METHOD M_InputMapping
VAR_INPUT
END_VAR
// TurnTable Axis sensor
arAxisCtrl_gb[AxisNo.TurnTable].SetupMode.bHomeSignal := NOT GVL_Input.uniDI.stDI.bTurnTable_Axis_HomeSensor;
// RoundBelt Axis sensor
arAxisCtrl_gb[AxisNo.RoundBelt].SetupMode.bHomeSignal := GVL_Input.uniDI.stDI.bRoundBelt_Axis_HomeSensor;
// Allocate Robot X Axis
arAxisCtrl_gb[AxisNo.Allocate_X].SetupMode.bPosLimitSignal:= NOT GVL_Input.uniDI.stDI.bAllocateRobot_Xaxis_PosLimit;
arAxisCtrl_gb[AxisNo.Allocate_X].SetupMode.bNegimitSignal:=  NOT GVL_Input.uniDI.stDI.bAllocateRobot_Xaxis_NegLimit;

//arAxisCtrl_gb[AxisNo.Allocate_Y].SetupMode.bHomeSignal:= ;
	//arAxisCtrl_gb[AxisNo.Allo cate_Y].SetupMode.bNegimitSignal:=;

arAxisCtrl_gb[AxisNo.OutRobot_X].SetupMode.bHomeSignal:= GVL_Input.uniDI.stDI.bOutRobot_Xaxis_HomeSensor;
arAxisCtrl_gb[AxisNo.OutRobot_X].SetupMode.bPosLimitSignal:=  NOT GVL_Input.uniDI.stDI.bOutRobot_Xaxis_PosLimit;
arAxisCtrl_gb[AxisNo.OutRobot_X].SetupMode.bNegimitSignal:=  NOT GVL_Input.uniDI.stDI.bOutRobot_Xaxis_NegLimit;

arAxisCtrl_gb[AxisNo.OutRobot_Y].SetupMode.bHomeSignal:= GVL_Input.uniDI.stDI.bOutRobot_Yaxis_HomeSensor;
arAxisCtrl_gb[AxisNo.OutRobot_Y].SetupMode.bPosLimitSignal:=  NOT GVL_Input.uniDI.stDI.bOutRobot_Yaxis_PosLimit;
arAxisCtrl_gb[AxisNo.OutRobot_Y].SetupMode.bNegimitSignal:=  NOT GVL_Input.uniDI.stDI.bOutRobot_Yaxis_NegLimit;

arAxisCtrl_gb[AxisNo.RackMotor].SetupMode.bNegimitSignal := NOT GVL_Input.uniDI.stDI.bStackPush_DCMotor_NegLimit;
arAxisCtrl_gb[AxisNo.RackMotor].SetupMode.bPosLimitSignal := not GVL_Input.uniDI.stDI.bStackPush_DCMotor_PosLimit;
END_METHOD

END_PROGRAM

// ---- Library/00_PackML/01_ObjectBase/FB_ModeBase_V1.TcPOU
(* the functionblock FB_ObjectBase_V1 is transmitted to every machineunit
*)
FUNCTION_BLOCK FB_ModeBase_V1 IMPLEMENTS ITF_UnitState
VAR_INPUT
    eModeCommand : DINT; //Mode from superior Unit
    eCommand     : E_PMLCommand := ePMLCommand_Abort; //Command for a new state from superior unit
	PackTag : Reference TO ST_PackMLv30;
END_VAR
VAR_OUTPUT
    eMode                  : DINT; //Actual mode of the Unit
    eState                 : E_PMLState (*:= ePMLState_Aborted*) ; //Actual state of the Unit
    bUndefinedDone         : BOOL; //When the SPS is started, the first state is Undefiend. bUndefined is TRUE, when the method Undefined has succesful finished
    bInvalidModeCommandOut : BOOL;
    bChangeIntoProduction  : BOOL;
END_VAR
VAR
    fbUnitModeManager : PML_UnitModeManager; //The PML_UnitModeManager manage the Modechanges
    fbStateMachine    : PML_StateMachine; //The PML_StateMachine mangae the Statechanges

    nStateModeChange : INT := 0; //Variable to handle the modechange
    nLastState       : E_PMLState; //Variable to store last state
END_VAR

CASE nStateModeChange OF
0:
	//Waiting for user request
	bChangeIntoProduction:= FALSE;
	IF  bButtonProductionReq AND (PackTag.Command.UnitMode = ePMLProtUnitMode_Production) AND (PackTag.Status.UnitModeCurrent = ePMLProtUnitMode_Invalid) THEN
			nStateModeChange	:= 1;
	ELSIF  PackTag.Command.UnitModeChangeRequest AND (PackTag.Command.UnitMode <> ePMLProtUnitMode_Production) THEN
			nStateModeChange	:= 1;
	ELSIF  bButtonProductionReq AND (PackTag.Command.UnitMode = ePMLProtUnitMode_Production) AND (PackTag.Status.UnitModeCurrent <> ePMLProtUnitMode_Production) THEN
			nStateModeChange	:= 3;
	END_IF
1:
	//Starting UnitModeManager 
	fbUnitModeManager.bExecute				:= TRUE;
	fbUnitModeManager.eModeCommand			:= eModeCommand;
	PackTag.Status.UnitModeChangeInProcess	:= TRUE;

	IF fbUnitModeManager.bDone THEN
		fbUnitModeManager.bExecute	:= FALSE;
		bInvalidModeCommandOut		:= FALSE;
		nStateModeChange			:= 0;
		bChangeIntoProduction		:= FALSE;
		
		PackTag.Status.UnitModeChangeInProcess	:= FALSE;
	ELSIF fbUnitModeManager.bError THEN
		bInvalidModeCommandOut		:= TRUE;
		fbUnitModeManager.bExecute	:= FALSE;
		
		nLastState					:= PackTag.Status.StateCurrent;
		nStateModeChange			:= 2;
		bChangeIntoProduction		:= FALSE;
		PackTag.Status.UnitModeChangeInProcess	:= FALSE;
	END_IF
2:
	//ErrorHanddling
	IF  PackTag.Command.UnitModeChangeRequest THEN
		nStateModeChange:=0;
		bInvalidModeCommandOut		:= FALSE;
	ELSIF nLastState<> PackTag.Status.StateCurrent THEN
		bInvalidModeCommandOut		:= FALSE;
	END_IF
	
3:
	//state to check, if command 'Porduction' is valid
	IF (PackTag.Status.StateCurrent = ePMLState_Aborted OR PackTag.Status.StateCurrent = ePMLState_Stopped OR PackTag.Status.StateCurrent = ePMLState_Idle) THEN
		bChangeIntoProduction		:= TRUE;
		IF stChangeIntoProduction.bYes OR stChangeIntoProduction.bYesReset THEN
			nStateModeChange			:= 1;		
		ELSIF stChangeIntoProduction.bNo THEN
			nStateModeChange			:= 0;
		END_IF
	ELSE
		nStateModeChange:= 2;
		bInvalidModeCommandOut		:= TRUE;
		nLastState					:= PackTag.Status.StateCurrent;
	END_IF
END_CASE


fbUnitModeManager(									
	eState			:= eState,
	eModeStatus		=> eMode,
	bDone			=> ,
	bError			=> ,
	nErrorId		=> );


IF fbUnitModeManager.eModeStatus <>  0 THEN
	//Calling the StateMachine, when there is a valid Mode
	fbStateMachine(
		eMode				:= eMode, 				
		eCommand			:= eCommand,			
		stSubUnitInfoRef	:= ,
		stOptions			:= , 
		eState				=> eState, 				
		bError				=> , 
		nErrorID			=> );
END_IF

//One of the methods is executing  by the actual state
CASE eState OF
	ePMLState_Undefined:
		M_Undefined();
	ePMLState_Clearing:
		M_Clearing();
	ePMLState_Stopped:
		M_Stopped();
	ePMLState_Starting:
		M_Starting();
	ePMLState_Idle:
		M_Idle();
	ePMLState_Suspended:
		M_Suspended();
	ePMLState_Execute:
		M_Execute();
	ePMLState_Stopping:
		M_Stopping();
	ePMLState_Aborting:
		M_Aborting();
	ePMLState_Aborted:
		M_Aborted();
	ePMLState_Holding:
		M_Holding();
	ePMLState_Held:
		M_Held();
	ePMLState_Unholding:
		M_Unholding();
	ePMLState_Suspending:
		M_Suspending();
	ePMLState_Unsuspending:
		M_Unsuspending();
	ePMLState_Resetting:
		M_Resetting();
	ePMLState_Completing:
		M_Completing();
	ePMLState_Complete:
		M_Complete();
END_CASE

{attribute 'object_name' := 'M_Aborted'}
METHOD M_Aborted
VAR_INPUT
END_VAR
M_StateComplete();
END_METHOD

{attribute 'object_name' := 'M_Aborting'}
METHOD M_Aborting
VAR_INPUT
END_VAR
M_StateComplete();
END_METHOD

{attribute 'object_name' := 'M_Clearing'}
METHOD M_Clearing
VAR_INPUT
END_VAR
M_StateComplete();
END_METHOD

{attribute 'object_name' := 'M_Complete'}
METHOD M_Complete
VAR_INPUT
END_VAR
M_StateComplete();
END_METHOD

{attribute 'object_name' := 'M_Completing'}
METHOD M_Completing
VAR_INPUT
END_VAR
M_StateComplete();
END_METHOD

{attribute 'object_name' := 'M_Execute'}
METHOD M_Execute
VAR_INPUT
END_VAR
M_StateComplete();
END_METHOD

{attribute 'object_name' := 'M_Held'}
METHOD M_Held
VAR_INPUT
END_VAR
M_StateComplete();
END_METHOD

{attribute 'object_name' := 'M_Holding'}
METHOD M_Holding
VAR_INPUT
END_VAR
M_StateComplete();
END_METHOD

{attribute 'object_name' := 'M_Idle'}
METHOD M_Idle
VAR_INPUT
END_VAR
M_StateComplete();
END_METHOD

{attribute 'object_name' := 'M_Resetting'}
METHOD M_Resetting
VAR_INPUT
END_VAR
M_StateComplete();
END_METHOD

{attribute 'object_name' := 'M_Starting'}
METHOD M_Starting
VAR_INPUT
END_VAR
M_StateComplete();
END_METHOD

{attribute 'object_name' := 'M_StateComplete'}
METHOD M_StateComplete
VAR_INPUT
END_VAR
//the actual state is completed
fbStateMachine.M_StateComplete();
END_METHOD

{attribute 'object_name' := 'M_Stopped'}
METHOD M_Stopped
VAR_INPUT
END_VAR
M_StateComplete();
END_METHOD

{attribute 'object_name' := 'M_Stopping'}
METHOD M_Stopping
VAR_INPUT
END_VAR
M_StateComplete();
END_METHOD

{attribute 'object_name' := 'M_Suspended'}
METHOD M_Suspended
VAR_INPUT
END_VAR
M_StateComplete();
END_METHOD

{attribute 'object_name' := 'M_Suspending'}
METHOD M_Suspending
VAR_INPUT
END_VAR
M_StateComplete();
END_METHOD

{attribute 'object_name' := 'M_Undefined'}
METHOD M_Undefined
VAR_INPUT
END_VAR
//bUndefinedDone := TRUE;
M_StateComplete();
END_METHOD

{attribute 'object_name' := 'M_Unholding'}
METHOD M_Unholding
VAR_INPUT
END_VAR
M_StateComplete();
END_METHOD

{attribute 'object_name' := 'M_Unsuspending'}
METHOD M_Unsuspending
VAR_INPUT
END_VAR
M_StateComplete();
END_METHOD

END_FUNCTION_BLOCK

// ---- Library/20_MachineUnits/21_StorageArea/Service/FB_LowerFeedInConveyor.TcPOU
FUNCTION_BLOCK FB_LowerFeedInConveyor EXTENDS FB_ActionBasic
VAR_INPUT
    xExecute    : BOOL;
    xAbort      : BOOL;
	xReset		: BOOL;
    Cylinder 	: REFERENCE TO UNI_CylinderList;
    TimeOut  	: LREAL := 30; // Unit : s
	Input		: ST_InputTable;
	OutPut		: ST_OutputTable;
	Motor		: REFERENCE TO UNI_MotorList;
END_VAR	
VAR_OUTPUT
    xAborted : BOOL;
    iErrorID : INT;
    ErrorMsg : T_MaxString;
END_VAR
VAR
    StateBehaviour   : CBML.ETrigATo;
    CurrentPosition : ST_PositionTable;
	uiCyclicStep    : UINT := 0;
	Reset_Rtrig 	:R_TRIG;
	
	TON_SensorDelay :TON;
	TON_ArrivedTimeOut :TON;
	TON_TimeOut :TON;
	fbExecuteEdgeDetect :FB_EdgeDetect;
END_VAR

THIS^.IBehaviourModel := StateBehaviour;
StateBehaviour(xExecute := xExecute,
              xAbort := xAbort OR fbExecuteEdgeDetect.xFallingEdge,
              udiTimeOut := LREAL_TO_UDINT( TimeOut*1000000),
              xDone => xDone,
              xBusy => xBusy,
              xError => xError,
              xAborted => xAborted);
//Error Mes
iErrorID := StateBehaviour._model.iErrorID;
ErrorMsg := M_GetErrorMsg(xErrorID := iErrorID);  

//Make sure that C# turns off execute to shut down the service
fbExecuteEdgeDetect(xInput :=xExecute);

//Reset 
Reset_Rtrig(CLK:= xReset);
IF Reset_Rtrig.Q THEN
	StateBehaviour.ResetModel(xCommit:=xReset);
END_IF

//Action
A00_BaseUnits();

ACTION A00_BaseUnits:
TON_SensorDelay(PT:= T#500MS);
TON_ArrivedTimeOut(PT:=T#30S);
TON_TimeOut(PT:=T#10S);
END_ACTION

METHOD CleanupAction
VAR_INPUT
    xAbortProposed : BOOL;
    iErrorIDProposed: INT;
END_VAR
VAR_OUTPUT
    xComplete : BOOL := TRUE;
    xAbort: BOOL := xAbortProposed;
 	iErrorID : INT := iErrorIDProposed;
END_VAR
END_METHOD

METHOD CyclicAction
VAR_INPUT
    itfTimingController : CBML.ITimingController;
END_VAR
VAR_OUTPUT
    xComplete : BOOL := TRUE;
    iErrorID : INT := 0;
END_VAR
xComplete :=FALSE;

CASE uiCyclicStep OF 
	
	100:	//檔盒上升， 呼叫輸送帶
		TON_TimeOut.IN:= TRUE;
		Cylinder.List.fbLowCV_Block2.M_Extend();
		IF Cylinder.List.fbLowCV_Block2.InFrontPosition THEN
			TON_TimeOut.IN:=FALSE;
			Motor.List.LowCV.M_MoveForward();
			uiCyclicStep:=150;
		END_IF
		IF TON_TimeOut.Q THEN 
			iErrorID :=10;
		END_IF
	150:	//check motor forward
		TON_TimeOut.IN :=TRUE;
		IF Motor.List.LowCV.InForWard THEN 
			TON_TimeOut.IN:=FALSE;
			uiCyclicStep:=200;
		END_IF
		IF TON_TimeOut.Q THEN
			iErrorID :=11;
		END_IF
	
	200:	//盒子到位, 延遲訊號,
		TON_ArrivedTimeOut.IN:= TRUE;
		TON_SensorDelay.IN := Input.bLowCV_Block2Detect_Sensor;
		IF TON_SensorDelay.Q THEN
			TON_SensorDelay.IN:=FALSE;
			TON_ArrivedTimeOut.IN:=FALSE;
			Cylinder.List.fbLowCV_Press4.M_Extend();
			uiCyclicStep:=300;
		END_IF
		IF TON_ArrivedTimeOut.Q THEN
			iErrorID :=9;
		END_IF
		
	300:	//檔盒下 等待第一盒到達最前sensor
		TON_TimeOut.IN:=TRUE;
		IF Cylinder.List.fbLowCV_Press4.InFrontPosition THEN
			Cylinder.List.fbLowCV_Block2.M_Retract();
		END_IF
		IF Cylinder.List.fbLowCV_Block2.InRearPosition THEN
			TON_TimeOut.IN:=FALSE;
			uiCyclicStep:=400;	
		END_IF
		IF TON_TimeOut.Q THEN
			iErrorID :=11;
		END_IF
		
	400:	//確認到最前sensor 
		TON_SensorDelay.IN:=Input.bLowCV_BoxArrived_Sensor;
		IF TON_SensorDelay.Q THEN
			TON_SensorDelay.IN:=FALSE;
			Cylinder.List.fbLowCV_Block2.M_Extend();
			uiCyclicStep:=500;
		END_IF
	
	500:	//釋放第二盒 
		IF 	Cylinder.List.fbLowCV_Block2.InFrontPosition THEN
			Cylinder.List.fbLowCV_Press4.M_Retract();
			uiCyclicStep:=600;
		END_IF
	600:	// 第二盒到檔盒位 第三盒壓盒檔上
		TON_SensorDelay.IN:= Input.bLowCV_Block2Detect_Sensor;
		IF TON_SensorDelay.Q THEN
			TON_SensorDelay.IN :=FALSE;
			Cylinder.List.fbLowCV_Press4.M_Extend();
			uiCyclicStep:= 700;
		END_IF
	
	700:	//釋放第二盒
		IF Cylinder.List.fbLowCV_Press4.InFrontPosition THEN
			Cylinder.List.fbLowCV_Block2.M_Retract();
			Cylinder.List.fbLowCV_Block1.M_Extend();
		END_IF
		IF Cylinder.List.fbLowCV_Block2.InRearPosition AND 
			Cylinder.List.fbLowCV_Block1.InFrontPosition THEN
			uiCyclicStep:= 800;
		END_IF
		
	800:	// 等待第二盒到夾盒位
		TON_SensorDelay.IN:=Input.bLowCV_Block1Detect_Sensor;
		IF TON_SensorDelay.Q THEN
			TON_SensorDelay.IN:=FALSE;
			Motor.List.LowCV.M_MotorStop();
			uiCyclicStep:=900;
		END_IF
	900:	//馬達停止 第一第二盒壓盒上
		IF Motor.List.LowCV.InStopped THEN
			Cylinder.List.fbLowCV_Press1.M_Extend();
			Cylinder.List.fbLowCV_Press2.M_Extend();
			Cylinder.List.fbLowCV_Block1.M_Retract();
			uiCyclicStep :=1000;
		END_IF
	1000:	//壓盒下
		IF Cylinder.List.fbLowCV_Press1.InFrontPosition AND 
			Cylinder.List.fbLowCV_Press2.InFrontPosition AND 
			Cylinder.List.fbLowCV_Block1.InRearPosition THEN
			Cylinder.List.fbLowCV_Press1.M_Retract();
			Cylinder.List.fbLowCV_Press2.M_Retract();
		END_IF
	1100:	//確認壓盒位置 回done
		IF Cylinder.List.fbLowCV_Press1.InRearPosition AND 
			Cylinder.List.fbLowCV_Press2.InRearPosition THEN 
			xComplete :=TRUE;
		END_IF
END_CASE
END_METHOD

METHOD ExitAction
VAR_INPUT
    xAfterCleanup : BOOL;
    xInCopyCode : BOOL;
END_VAR
TON_SensorDelay.IN:=FALSE;
END_METHOD

METHOD M_GetErrorMsg : T_MaxString
VAR_INPUT
	xErrorID: INT;
END_VAR

VAR
	
END_VAR
CASE xErrorID OF
	0:
		M_GetErrorMsg := 'No Error';
	1:
		M_GetErrorMsg := 'Action time out';
	2:
		M_GetErrorMsg := 'Position Data invalid';
	3:
		M_GetErrorMsg := 'LowCV_Block1 has Error in StartAction ';
	4:
		M_GetErrorMsg := 'LowCV_Block2 has Error in StartAction';
	5:
		M_GetErrorMsg := 'LowCV_Press1 has Error in StartAction';
	6:
		M_GetErrorMsg := 'LowCV_Press2 has Error in StartAction';
	7:
		M_GetErrorMsg := 'fbLowCV_Press3 has Error in StartAction';
	8:
		M_GetErrorMsg := 'fbLowCV_Press4 has Error in StartAction';
	9:
		M_GetErrorMsg := 'Box Arrived Time out not on LowCVBlock2' ;
	10:
		M_GetErrorMsg := 'Cylinder Error in CyclicAction';
	11:
		M_GetErrorMsg := 'Motor Error in CyclicAction';
									
		
		
		
		
END_CASE
END_METHOD

METHOD ResetAction
VAR_OUTPUT
    xComplete : BOOL := TRUE;
END_VAR
END_METHOD

METHOD StartAction
VAR_OUTPUT
    xComplete : BOOL := TRUE;
	iErrorID : INT := 0;
END_VAR
xComplete :=FALSE;

TON_SensorDelay.IN:=FALSE;

IF Cylinder.List.fbLowCV_Block1.xError THEN
	iErrorID := 3;
END_IF
IF Cylinder.List.fbLowCV_Block2.xError THEN
	iErrorID := 4;
END_IF
IF Cylinder.List.fbLowCV_Press1.xError THEN
	iErrorID := 5;
END_IF
IF Cylinder.List.fbLowCV_Press2.xError THEN
	iErrorID := 6;
END_IF
IF Cylinder.List.fbLowCV_Press3.xError THEN
	iErrorID := 7;
END_IF
IF Cylinder.List.fbLowCV_Press4.xError THEN
	iErrorID := 8;
END_IF

IF Cylinder.List.fbLowCV_Block1.InRearPosition AND
	Cylinder.List.fbLowCV_Block2.InRearPosition AND 
	Cylinder.List.fbLowCV_Press1.InRearPosition AND 
	Cylinder.List.fbLowCV_Press2.InRearPosition AND 
	Cylinder.List.fbLowCV_Press3.InRearPosition AND 
	Cylinder.List.fbLowCV_Press4.InRearPosition AND 
	Input.bLowCV_2ndBoxGap_Sensor THEN	//reverse logic sensor ,do make sure no box here 
	xComplete :=TRUE;
END_IF
END_METHOD

END_FUNCTION_BLOCK

// ---- Library/20_MachineUnits/22_AllocateArea/FB_AllocateAreaWithXPlanar.TcPOU
FUNCTION_BLOCK FB_AllocateAreaWithXPlanar EXTENDS FB_ModeBase_V1
VAR_INPUT
	
END_VAR
VAR_OUTPUT
END_VAR
VAR
	UnitInput :REFERENCE TO ST_AllocateInput;
	UnitOutput: REFERENCE TO ST_AllocateOutput;
END_VAR

{attribute 'object_name' := 'M_Aborted'}
METHOD M_Aborted 
VAR_INPUT
END_VAR
END_METHOD

{attribute 'object_name' := 'M_Aborting'}
METHOD M_Aborting
VAR_INPUT
END_VAR
END_METHOD

{attribute 'object_name' := 'M_Clearing'}
METHOD M_Clearing
VAR_INPUT
END_VAR
END_METHOD

{attribute 'object_name' := 'M_Complete'}
METHOD M_Complete
VAR_INPUT
END_VAR
END_METHOD

{attribute 'object_name' := 'M_Completing'}
METHOD M_Completing
VAR_INPUT
END_VAR
END_METHOD

{attribute 'object_name' := 'M_Execute'}
METHOD M_Execute
VAR_INPUT
END_VAR
M_StateComplete();
END_METHOD

{attribute 'object_name' := 'M_Held'}
METHOD M_Held
VAR_INPUT
END_VAR
END_METHOD

{attribute 'object_name' := 'M_Holding'}
METHOD M_Holding
VAR_INPUT
END_VAR
END_METHOD

{attribute 'object_name' := 'M_Idle'}
METHOD M_Idle
VAR_INPUT
END_VAR
END_METHOD

METHOD M_IOMapping
VAR_INPUT
END_VAR
//UnitInput := GVL_in
END_METHOD

{attribute 'object_name' := 'M_Resetting'}
METHOD M_Resetting
VAR_INPUT
END_VAR
END_METHOD

{attribute 'object_name' := 'M_Starting'}
METHOD M_Starting
VAR_INPUT
END_VAR
VAR
	uiStartingStep : DINT;
END_VAR
CASE eMode OF
    E_Mode.Auto:
        CASE uiStartingStep OF
            0: //
            1: //
            2: //
            3: //
            9900:
                M_StateComplete();
        END_CASE
END_CASE
END_METHOD

{attribute 'object_name' := 'M_Stopped'}
METHOD M_Stopped
VAR_INPUT
END_VAR
END_METHOD

{attribute 'object_name' := 'M_Stopping'}
METHOD M_Stopping
VAR_INPUT
END_VAR
END_METHOD

{attribute 'object_name' := 'M_Suspended'}
METHOD M_Suspended
VAR_INPUT
END_VAR
END_METHOD

{attribute 'object_name' := 'M_Suspending'}
METHOD M_Suspending
VAR_INPUT
END_VAR
END_METHOD

{attribute 'object_name' := 'M_Undefined'}
METHOD M_Undefined
VAR_INPUT
END_VAR
END_METHOD

{attribute 'object_name' := 'M_Unholding'}
METHOD M_Unholding
VAR_INPUT
END_VAR
END_METHOD

{attribute 'object_name' := 'M_Unsuspending'}
METHOD M_Unsuspending
VAR_INPUT
END_VAR
END_METHOD

END_FUNCTION_BLOCK

// ---- Library/99_Utilities/ErrorHandling/FB_ErrorHandler_OLD.TcPOU
{attribute 'reflection'}
FUNCTION_BLOCK PUBLIC FB_ErrorHandler_OLD IMPLEMENTS ITF_ErrorHandlerSubject
VAR_INPUT
END_VAR
VAR_OUTPUT
    astrActive : ARRAY [0..999] OF ST_Alarm_Tmax;	//State from all existing FB
	uiNumOfActError : UINT;	
	bErrorOccur 	:BOOL;
END_VAR
VAR
	
	//{attribute 'hide'}
	fbLocalSystemTime				: FB_LocalSystemTime := (bEnable := TRUE, dwCycle := 1);
    {attribute 'instance-path'} 
    {attribute 'noinit'}
    _strName: STRING(255); 					// Instance path of the FB for Diagnostic
			
	_stInfoState : ARRAY [1..GVL.MAX_Observer] OF ST_BehaviourInfo;	//State from all existing FB
	_stErrorState : ARRAY [1..GVL.MAX_Observer] OF BOOL;			//State from all existing FB
	_UniqueErrorCode : ARRAY [1..GVL.MAX_Observer] OF string;
	_uiNumberOfDevices : UINT;						//Number of Attached Devices
	uiHelp : INT; 									//Help Variable for Loop
	
	//Help Variables for Attaching and read Information from Devices
	aritfObserver : ARRAY [0..GVL.MAX_Observer]OF IBasicElement;
	uiLoop : UINT;
	uiErrorIndex : UINT;
    astrClear : ARRAY [0..999] OF ST_Alarm_Tmax;	//State from all existing FB
	_stErrorState_Clear : ARRAY [1..GVL.MAX_Observer] OF BOOL;			//State from all existing FB for clear	
	tonClearErrorDelay : TON;
	uiStep : UINT:=0;
	
END_VAR

_uiNumberOfDevices := 0;
fbLocalSystemTime();


tonClearErrorDelay(PT:=T#100MS);

CASE uiStep OF
	
0: //Init step
	tonClearErrorDelay.IN :=FALSE;
	bErrorOccur :=FALSE;
	uiStep :=100;
	
100: // Delay for a while
	tonClearErrorDelay.IN :=TRUE;
	IF tonClearErrorDelay.Q THEN
		uiStep := 300;
	END_IF
		
200: //Clear error
		astrActive := astrClear;
		_stErrorState :=_stErrorState_Clear;
		uiStep := 0;
300: //Working
FOR uiLoop := 0 TO GVL.MAX_Observer DO
    IF aritfObserver[uiLoop] <> 0 THEN

        _uiNumberOfDevices := _uiNumberOfDevices + 1;
        aritfObserver[uiLoop].GetModelState(
                xDone    => _stInfoState[uiLoop].xDone,
                xBusy    => _stInfoState[uiLoop].xBusy,
                xError   => _stInfoState[uiLoop].xError,
                xAborted => _stInfoState[uiLoop].xAborted,
                iErrorID => _stInfoState[uiLoop].iErrorID, 
				UniqueErrorCode =>_UniqueErrorCode[uiLoop]);

        _stInfoState[uiLoop].strName := aritfObserver[uiLoop].GetName();

        IF NOT _stErrorState[uiLoop] AND _stInfoState[uiLoop].xError THEN
            _stErrorState[uiLoop] := _stInfoState[uiLoop].xError;
			bErrorOccur :=TRUE;

            //Build Error String
            FOR uiHelp := 999 TO 0 BY -1 DO
                IF uiHelp > 0 THEN
                    // Sort the array down once, leaving the first row of the array empty.
                    astrActive[uiHelp] := astrActive[uiHelp - 1];
                ELSIF uiHelp = 0 THEN
                    astrActive[uiHelp].Message := CONCAT(
                            CONCAT(CONCAT('In FB ', _stInfoState[uiLoop].strName), ' the error is active : '),
                            FC_ErrorCode(_stInfoState[uiLoop].iErrorID));

                    astrActive[uiHelp].ID       := _stInfoState[uiLoop].iErrorID;
                    astrActive[uiHelp].Trigger  := _stInfoState[uiLoop].xError;
                    astrActive[uiHelp].DateTime := TIMESTRUCT_TO_PackMLTime(fbLocalSystemTime.systemTime);
					astrActive[uiHelp].UniqueErrorCode:=_UniqueErrorCode[uiLoop];
               		//astrActive[uiHelp].Value   :=	_UniqueErrorCode[uiLoop];
				 END_IF
            END_FOR
//        ELSIF _stErrorState[uiLoop] AND NOT _stInfoState[uiLoop].xError THEN
//            _stErrorState[uiLoop] := _stInfoState[uiLoop].xError;

//            //Build Error String
//            FOR uiHelp := 999 TO 0 BY -1 DO
//                IF uiHelp > 0 THEN
//                    astrActive[uiHelp] := astrActive[uiHelp - 1];
//                ELSIF uiHelp = 0 THEN
//                    astrActive[uiHelp].Message := CONCAT(
//                            CONCAT(CONCAT('In FB ', _stInfoState[uiLoop].strName), 'the following error is deactive:'),
//                            FC_ErrorCode(_stInfoState[uiLoop].iErrorID));
//                END_IF
//            END_FOR
        END_IF
		
	ELSE
	//	EXIT;	
    END_IF
END_FOR

END_CASE

METHOD AttachDevice 
(*Register a Device by the BehaiourModel Interface*)
VAR_INPUT
	(*Device which will be monitor from Error Handler*)
	IDevice	: IBasicElement;
END_VAR

VAR
	uiLoop: UINT;
END_VAR
FOR uiLoop := 1 TO GVL.MAX_Observer DO
	IF IDevice <> 0 AND THIS^.aritfObserver[uiLoop]= 0 THEN
		THIS^.aritfObserver[uiLoop] := IDevice;
		EXIT;
	END_IF
END_FOR
END_METHOD

METHOD ClearError
VAR_INPUT
END_VAR
astrActive := astrClear;
_stErrorState :=_stErrorState_Clear; // not necessary but keep it

uiStep := 200; // Go to clear error step
END_METHOD

METHOD DetachDevice 
(*Unregister a Device by the BehaiourModel Interface*)
VAR_INPUT
	(*Device which will be deleted from the monitor Error Handler list*)
	IDevice	: IBasicElement;
END_VAR

VAR
	uiLoop: UINT;
END_VAR
FOR uiLoop := 0 TO GVL.MAX_Observer DO
	IF IDevice <> 0 AND THIS^.aritfObserver[uiLoop]= IDevice THEN
		THIS^.aritfObserver[uiLoop] := 0;
		EXIT;
	END_IF
END_FOR
END_METHOD

END_FUNCTION_BLOCK

// ---- Library/99_Utilities/ErrorHandling/FB_ErrorHandler_abond.TcPOU
FUNCTION_BLOCK FB_ErrorHandler_abond EXTENDS FB_ActionBasic
VAR_INPUT
	xEnable : BOOL;
	stAdmin : REFERENCE TO ST_PMLa;
	AlarmList :REFERENCE TO ARRAY[0..999] OF ST_Alarm_Tmax;
END_VAR
VAR_OUTPUT
END_VAR
VAR
	StateBehavior : CBML.LConC;
	ErrorCount : DINT;
END_VAR

THIS^.IBehaviourModel := StateBehavior;
StateBehavior(xEnable:= xEnable, xBusy=> xBusy, xError=> xError);
//AlarmCtrl();
//IF btest THEN
//stAlarm.Trigger := TRUE;
//stAlarm.Message := 'test';
//AlarmCtrl.M_SetAlarm(stAdmin := GVL_Machine.PackTags[0].Admin, stAlarm := stAlarm);
//END_IF

METHOD CleanupAction
VAR_INPUT
    xAbortProposed : BOOL;
    iErrorIDProposed: INT;
END_VAR
VAR_OUTPUT
    xComplete : BOOL := TRUE;
    xAbort: BOOL := xAbortProposed;
 	iErrorID : INT := iErrorIDProposed;
END_VAR
END_METHOD

METHOD CyclicAction
VAR_INPUT
    itfTimingController : CBML.ITimingController;
END_VAR
VAR_OUTPUT
    xComplete : BOOL := TRUE;
    iErrorID : INT := 0;
END_VAR
VAR
	diCheckTriggerLoop : DINT;
	diCheckAlarmLoop : DINT;
	bHasSameID :BOOL;
END_VAR
VAR_INST
	diSearchID : DINT;
END_VAR
xComplete := FALSE;
bHasSameID := FALSE;
diSearchID := 0;
FOR diCheckTriggerLoop := 1 TO stAdmin.AlarmExtent DO
    IF stAdmin.Alarm[diCheckTriggerLoop].Trigger THEN
        FOR diCheckAlarmLoop := 0 TO 999 DO
            IF AlarmList[diCheckAlarmLoop].ID = stAdmin.Alarm[diCheckTriggerLoop].ID THEN
				diSearchID := diCheckTriggerLoop;
                bHasSameID := TRUE;
				EXIT;
            END_IF
        END_FOR
    END_IF

    IF NOT bHasSameID THEN
        ErrorCount := ErrorCount + 1;
        AlarmList[ErrorCount].ID := DINT_TO_UDINT(stAdmin.Alarm[diCheckTriggerLoop].ID);
        AlarmList[ErrorCount].Category := stAdmin.Alarm[diCheckTriggerLoop].Category;
        AlarmList[ErrorCount].Message := stAdmin.Alarm[diCheckTriggerLoop].Message;
        AlarmList[ErrorCount].Value := stAdmin.Alarm[diCheckTriggerLoop].Value;
        AlarmList[ErrorCount].Trigger := stAdmin.Alarm[diCheckTriggerLoop].Trigger;
    END_IF
END_FOR
END_METHOD

METHOD ExitAction
VAR_INPUT
    xAfterCleanup : BOOL;
    xInCopyCode : BOOL;
END_VAR
END_METHOD

METHOD ResetAction
VAR_OUTPUT
    xComplete : BOOL := TRUE;
END_VAR
END_METHOD

METHOD StartAction
VAR_OUTPUT
    xComplete : BOOL := TRUE;
	iErrorID : INT := 0;
END_VAR
END_METHOD

END_FUNCTION_BLOCK

// ---- Library/99_Utilities/ErrorHandling/FB_ErrorHandling.TcPOU
FUNCTION_BLOCK FB_ErrorHandling
VAR_INPUT
	xEnable : BOOL := TRUE;
	tInitBypassDelayTime : TIME;
END_VAR

VAR_OUTPUT
	xError		: BOOL; // Normal Error -> Go to Held
	//xFatalError : BOOL; // Fatal Error -> Go to Abort
	xWarning	: BOOL; // System have warning
	xSeverity : E_Severity;
END_VAR

VAR
	bFirstCycle			: BOOL := TRUE;
	bCoresysError		: BOOL; // At least one Coresys has an error 
	bXTSError			: BOOL; // At least one XTS has an error 
	dwXTSDiagNo			: DWORD; // XTS diag number
	strXTSDiagMessage : STRING(60); // XTS diag text
	uiXTSSeverity		: UINT; // XTS error severity
	bAppError			: BOOL; // User defined error
	bECatError			: BOOL; // EtherCAT module error
	dwAppDiagNo			: DWORD; // User diag number
	strAppDiagMessage : STRING(60); // User diag text
	uiAppErrSeverity	: UINT; // User error severity
	bSubsysError		: BOOL; // Subsys has an error
	// FB_AnyAborted_Rtrig : R_TRIG ;
	udiErrorCount					: UDINT;
	fbMachineCtrlInitDOne_Rtrig		: R_TRIG;
	fbMachineResetBtn_FTrig			: F_TRIG;
	bClearEthercatErr				: BOOL; // 臨時版本
	udiIndex						: UDINT;
	bAnySubAborted					: BOOL; // Currently, there is at least one Sub station in an aborted state.
	bST01_Alarm						: BOOL;
	bST03_Alarm						: BOOL;
	bST06_Alarm						: BOOL;
	bST10_Alarm						: BOOL;
	bST12_Alarm						: BOOL;
	bST14_Alarm						: BOOL;
	bST15_Alarm						: BOOL;
	bST17_Alarm						: BOOL;
	bST18_Alarm						: BOOL;
	bST20_Alarm						: BOOL;
	bST22_Alarm						: BOOL;
	bST23_Alarm						: BOOL;
	bST25_Alarm						: BOOL;
	bST27_Alarm						: BOOL;
	bST30_Alarm						: BOOL;
	bXTSShuttleError				: BOOL;
	bXTSModuleError					: BOOL;
	bXTSNcError						: BOOL;
	bResetRetry						: BOOL;
	TON_ResetRetry					: TON;
	FB_CoresysErrorHandler			: FB_CoresysErrorHandler;
	TON_ClearDelayCheck				: TON;
	bSubsysWarning					: BOOL;
	Ton_InitBypassDelay				: TON;
	FB_EtherCATErrorHandler			: FB_EtherCATErrorHandler;
	arrUnitsWarningHandler			: ARRAY[1..cudiXTS_MaxIndex]OF FB_AppWarningHandler;
	I_UnitsWarningHandler			: ARRAY[1..cudiXTS_MaxIndex]OF ITF_SubUnitWarning;
	TON_KeepMDSError 				: TON;
	TON_CheckMDSNoError				: TON;
	bCheckMDSError					: BOOL;
	TOF_KeepMDSError_Delay			: TOF;

END_VAR

Ton_InitBypassDelay(PT:= T#5S);
IF NOT xEnable THEN
	RETURN;
ELSIF ( bFirstCycle = TRUE ) THEN
	Ton_InitBypassDelay.IN := TRUE;
	M_OneTimeInit();
	RETURN;
END_IF


//TON_ClearDelayCheck(IN := bClearbyPassDelay, PT := T#800MS);

//IF TON_ClearDelayCheck.Q THEN
//	bClearbyPassDelay := FALSE;
//END_IF

//IF bReset_gb THEN
//	THIS^.M_Reset();
//END_IF
//IF   NOT FB_Safety.bSafetyOK AND_THEN M_FindMDSError() THEN
//	bKeepMDSError := TRUE;
//END_IF
//TON_KeepMDSError(IN := bKeepMDSError,PT := T#3S);
//bCheckMDSError := FALSE;
//FOR udiIndex := 1 TO UDINT_TO_UINT(udiMax_MachineAlarm_Index) DO
//	IF PackTags.Machine.Admin.Alarm[udiIndex].ID = DINT#990281 THEN
//		bCheckMDSError := TRUE;
//	END_IF
//END_FOR
//TON_CheckMDSNoError(IN := (NOT FB_MDS.bMoverIdDetectionError) AND (NOT FB_MDS.bError) AND (NOT bCheckMDSError), PT := T#1S  );
//TOF_KeepMDSError_Delay(IN:= TON_CheckMDSNoError.Q ,PT:=T#2S);

//IF  TOF_KeepMDSError_Delay.Q THEN
//	bKeepMDSError := false;
//END_IF
// Alarm Histroy Upload
M_UploadData();
//------------------------------------------------------------------------------------------------------
//------------------------------------- Scan errors  ---------------------------------------------------  
//------------------------------------------------------------------------------------------------------
M_ScanError();

M_ErrorAction(xSeverity=> xSeverity);

ACTION EtherCAT_Diag:
fbMachineCtrlInitDOne_Rtrig(CLK := bMachineCtrlInitDOne);
fbMachineResetBtn_FTrig(CLK := bReset_gb);

IF fbMachineCtrlInitDOne_Rtrig.Q OR fbMachineResetBtn_FTrig.Q THEN
	FOR udiIndex := 1 TO TO_UDINT(udiECatMasterNum) DO
		// Check mapping status
		IF (F_GetMappingStatus(p := ADR(arruiFrm0WcStateMapping[udiIndex]), n := SIZEOF(arruiFrm0WcStateMapping[udiIndex]))
			= EPlcMappingStatus.MS_Mapped)
			OR (
			F_GetMappingStatus(p := ADR(arruiFrm0WcStateMapping[udiIndex]), n := SIZEOF(arruiFrm0WcStateMapping[udiIndex]))
			= EPlcMappingStatus.MS_Partial)
			THEN
			arrfbEtherCatDiagnostics[udiIndex].bEnable := TRUE;
		END_IF
	END_FOR
END_IF

// 臨時版本
IF bClearEthercatErr THEN
	FOR udiIndex := 1 TO TO_UDINT(udiECatMasterNum) DO
		// Check mapping status
		IF (F_GetMappingStatus(p := ADR(arruiFrm0WcStateMapping[udiIndex]), n := SIZEOF(arruiFrm0WcStateMapping[udiIndex]))
			= EPlcMappingStatus.MS_Mapped)
			OR (
			F_GetMappingStatus(p := ADR(arruiFrm0WcStateMapping[udiIndex]), n := SIZEOF(arruiFrm0WcStateMapping[udiIndex]))
			= EPlcMappingStatus.MS_Partial)
			THEN
			arrfbEtherCatDiagnostics[udiIndex].bEnable := FALSE;
		END_IF
	END_FOR

	bClearEthercatErr := FALSE;
END_IF

// FB_EtherCatDiagnostics
FOR udiIndex := 1 TO TO_UDINT(udiECatMasterNum) DO
	// Check mapping status
	IF (F_GetMappingStatus(p := ADR(arruiFrm0WcStateMapping[udiIndex]), n := SIZEOF(arruiFrm0WcStateMapping[udiIndex]))
		= EPlcMappingStatus.MS_Mapped)
		OR (F_GetMappingStatus(p := ADR(arruiFrm0WcStateMapping[udiIndex]), n := SIZEOF(arruiFrm0WcStateMapping[udiIndex]))
		= EPlcMappingStatus.MS_Partial)
		THEN
		arrfbEtherCatDiagnostics[udiIndex](uiFrm0WcStateMapping := arruiFrm0WcStateMapping[udiIndex],
											uiFrm1WcStateMapping := arruiFrm1WcStateMapping[udiIndex],
											uiFrm2WcStateMapping := arruiFrm2WcStateMapping[udiIndex],
											uiFrm3WcStateMapping := arruiFrm3WcStateMapping[udiIndex],
											wDeviceIDMapping := arrwDeviceIDMapping[udiIndex],
											bEnable :=,
											pstDiagnosticResult := ADR(arrstDiagnosticResult[udiIndex]),
											pstFuncBlocksErr := ADR(arrstFuncBlocksErr[udiIndex]),
											bBusy =>,
											bActive =>,
											bError =>);
	END_IF
END_FOR
END_ACTION

METHOD FB_exit : BOOL
VAR_INPUT
	bInCopyCode : BOOL; // if TRUE, the exit method is called for exiting an instance that is copied afterwards (online change).
END_VAR
// 避免再切config時出現動態記憶體異常
fbAlarmTrigList.releaseQueue();
fbAlarmResetList.releaseQueue();
END_METHOD

METHOD GetAbort : BOOL
VAR_INPUT
END_VAR
VAR
	// Subsys Station number
	udiSubIndex : UDINT;
END_VAR
VAR_OUTPUT
	xErrorID : UDINT;
	//	ErrorMsg: STRING(255);
END_VAR
GetAbort := FALSE;

FOR udiSubIndex := 1 TO cudiXTS_MaxIndex DO
	IF (PackTags.arrSubSys_Station^[udiSubIndex].Status.StateCurrent = ePMLState_Aborted)
		AND (stSysParameters_Current.arIndexProductionValid[udiSubIndex] = E_ProductionValid.Valid)
		THEN
		xErrorID := 1100 + udiSubIndex;
		//FB_AppErrorHandler.M_SetAlarm(xUnitName := FB_AppErrorHandler.GetName(), xErrorID := xErrorID);
		GetAbort := TRUE;
		RETURN;

	END_IF
END_FOR

IF (PackTags.XTS.Status.StateCurrent = ePMLState_Aborted) THEN
	xErrorID := 1100;
	//FB_AppErrorHandler.M_SetAlarm(xUnitName := FB_AppErrorHandler.GetName(), xErrorID := xErrorID);
	GetAbort := TRUE;
END_IF
END_METHOD

METHOD GetHeld : BOOL
VAR_INPUT
END_VAR
VAR
	// Subsys Station number
	udiSubIndex : UDINT;
END_VAR
GetHeld := FALSE;

FOR udiSubIndex := 1 TO cudiXTS_MaxIndex DO
	IF (PackTags.arrSubSys_Station^[udiSubIndex].Status.StateCurrent = ePMLState_Held) THEN
		GetHeld := TRUE;
	END_IF
END_FOR

IF (PackTags.XTS.Status.StateCurrent = ePMLState_Held) THEN
	GetHeld := TRUE;
END_IF
END_METHOD

METHOD M_CoresysErrorHandle
VAR_INPUT
END_VAR
VAR
	udiLoop : UDINT;
	xarObserver		: ARRAY[1..MAX_Observer] OF ST_Alarm;
END_VAR
VAR_INST
	xErrorFound : BOOL;
END_VAR
VAR_OUTPUT
	xError : BOOL;
END_VAR
//IF bMachineCtrlInitDOne THEN
	FB_CoresysErrorHandler(xError=>xError);
//END_IF
END_METHOD

METHOD M_ErrorAction
VAR_INPUT
END_VAR

VAR
	udiLoop: UDINT;
END_VAR
VAR_INST
	bSafetyDoorOpened : BOOL;
END_VAR
VAR_OUTPUT
	xSeverity : E_Severity;
END_VAR
//xSeverity := 0;
//FOR udiLoop := 1 TO udiMax_MachineAlarm_Index DO
//	IF PackTags.Machine.Admin.Alarm[udiLoop].Value > xSeverity THEN
//		xSeverity := PackTags.Machine.Admin.Alarm[udiLoop].Value;
//	END_IF
//END_FOR
//bSafetyDoorOpened := FALSE;
//FOR udiLoop := 1 TO cgudiNumOfSafetyDoor DO
//	IF arrSafetyDoorStatus[udiLoop].bButton THEN
//		bSafetyDoorOpened := TRUE;
//		EXIT;
//	END_IF
//END_FOR
//IF ( xSeverity = E_Severity.Level7 ) THEN
//	IF xError
//		AND NOT ((PackTags.Machine.Status.StateCurrent=ePMLState_Aborted) 
//		OR (PackTags.Machine.Status.StateCurrent=ePMLState_Aborting) 
//		OR (PackTags.Machine.Status.StateCurrent = ePMLState_Clearing))
//	THEN
//		PackTags.Machine.Command.CntrlCmd := ePMLCommand_Abort;
//		PackTags.Machine.Command.CmdChangeRequest := TRUE;
//	END_IF
//ELSIF xSeverity = E_Severity.Level6 THEN
//	IF xError THEN
//		IF (PackTags.Machine.Status.StateCurrent= ePMLState_Execute AND NOT ((PackTags.Machine.Status.UnitModeCurrent = E_MachineMode.Manual) AND bSafetyDoorOpened) )
//			OR  (PackTags.Machine.Status.StateCurrent= ePMLState_Suspended)
//			OR  (PackTags.Machine.Status.StateCurrent= ePMLState_Unsuspending)
//			OR  (PackTags.Machine.Status.StateCurrent= ePMLState_Suspending)
//			OR  (PackTags.Machine.Status.StateCurrent= ePMLState_Held)
//			OR  (PackTags.Machine.Status.StateCurrent= ePMLState_Unholding)
//			OR  (PackTags.Machine.Status.StateCurrent= ePMLState_Holding) 
//		THEN
//		PackTags.Machine.Command.CntrlCmd := ePMLCommand_Hold;
//		PackTags.Machine.Command.CmdChangeRequest := TRUE;
//		ELSIF (PackTags.Machine.Status.UnitModeCurrent = E_MachineMode.Manual) AND bSafetyDoorOpened
//				AND NOT FB_MDS.bAllShuttlesNotMoving
////				AND NOT (PackTags.XTS.Status.StateCurrent = ePMLState_Aborted)
////				AND NOT (PackTags.XTS.Status.StateCurrent = ePMLState_Aborting)
////				AND NOT (PackTags.XTS.Status.StateCurrent = ePMLState_Clearing)
//		THEN
//		PackTags.XTS.Command.CntrlCmd := ePMLCommand_Abort;
//		PackTags.XTS.Command.CmdChangeRequest := TRUE;
//		END_IF
//	END_IF
//ELSIF xSeverity = E_Severity.Level5 THEN
//	IF xError THEN
//		IF (PackTags.Machine.Status.StateCurrent= ePMLState_Execute)
//			AND (PackTags.Machine.Status.UnitModeCurrent = E_MachineMode.Initialization)
//		THEN
//		PackTags.Machine.Command.CntrlCmd := ePMLCommand_Stop;
//		PackTags.Machine.Command.CmdChangeRequest := TRUE;
//		END_IF
//	END_IF
//END_IF
END_METHOD

METHOD M_EtherCATErrorHandler
VAR_INPUT
END_VAR
VAR_OUTPUT
	xError:BOOL;
END_VAR
//THIS^.xError := FALSE;
FOR udiIndex := 1 TO udiECatMasterNum DO
	arFB_ECatDiag[udiIndex](udiEcDeviceIndex:=udiIndex,xError=>);
	IF arFB_ECatDiag[udiIndex].xError THEN
		xError :=TRUE;
	END_IF
END_FOR
END_METHOD

METHOD M_FindMDSError : BOOL
VAR_INPUT
END_VAR
VAR
	udiAlarmIndex : UDINT;
END_VAR
FOR udiAlarmIndex := 1 TO udiMax_MachineAlarm_Index DO
	IF PackTags.Machine.Admin.Alarm[udiAlarmIndex].ID = DINT#990281 THEN
		M_FindMDSError := TRUE;
	END_IF
END_FOR
END_METHOD

METHOD M_OneTimeInit
VAR_INPUT
END_VAR

IF Ton_InitBypassDelay.Q THEN
	bFirstCycle := FALSE;
	Ton_InitBypassDelay.IN := FALSE;
END_IF
END_METHOD

METHOD M_Reset
VAR_INPUT
END_VAR
//// Clear Safety error.
//IF FB_Safety.stSafetyMapping.stSafetyProject.stGroupInput.bInRun
//	AND NOT bEStopActived_gb THEN
//	FB_Safety.reset();
//END_IF

//// XTS motion calculation
//IF fbXTSCalc.bError THEN
//	fbXTSCalc.M_Reset();
//END_IF


//IF FB_XTS.FB_InitializationMode.xError THEN
//	FB_XTS.FB_InitializationMode.M_ClearStatus();
//END_IF

//IF fbShuttlesConsvNGMon.bError THEN
//	fbShuttlesConsvNGMon.M_Reset();
//END_IF



//IF FB_CoreSys_gb.FB_Machine_ProductionMode.xError THEN
//	FB_CoreSys_gb.FB_Machine_ProductionMode.M_ClearError();
//END_IF


//IF FB_CoreSys_gb.FB_Machine_InitializationMode.xError THEN
//	FB_CoreSys_gb.FB_Machine_InitializationMode.M_ClearError();
//END_IF


//IF FB_LubricationCamPnp.Error THEN
//	FB_LubricationCamPnp.Reset();
//END_IF

//IF FB_LubricationXTS.Error THEN
//	FB_LubricationXTS.Reset();
//END_IF
	

//IF FB_HealthBit_HMI.bError THEN
//	FB_HealthBit_HMI.M_Reset();
//END_IF

//IF FB_IPCShutDown.bError THEN
//	FB_IPCShutDown.M_Reset();
//END_IF 		

//IF FB_IPCPowerFailureHandler.bError THEN
//	FB_IPCPowerFailureHandler.M_Reset();
//END_IF

//IF FB_Reset_Rtrig.Q AND FB_DataRecovery.bError THEN
//	FB_DataRecovery.M_Reset();
//END_IF 

//IF FB_Reset_Rtrig.Q AND fbTerminateBatch.bError THEN
//	fbTerminateBatch.M_Reset();
//END_IF

//IF bECatError THEN
//	bECatError := FALSE;
//END_IF
END_METHOD

METHOD M_ScanError
VAR_INPUT
END_VAR

VAR
	udiLoop : UDINT;
END_VAR
VAR_INST
	bECatError_Mem : BOOL;
END_VAR
// Ethercat Diag
EtherCAT_Diag();
//FB_EtherCATErrorHandler(xError=>bECatError);
M_EtherCATErrorHandler(xError =>bECatError_Mem);
IF  bECatError_Mem THEN
	bECatError := TRUE;
END_IF
// XTS error combinations.
M_XTSErrorHandle();

// Coresys error combinations.
M_CoresysErrorHandle(xError=> bAppError);
bCoresysError := bXTSError OR bAppError OR bECatError;

// Subsys error combinations

M_SubsysErrorHandle(xError => bSubsysError);
//M_SubsysWarrningHandle(xWarning => bSubsysWarning);
M_SubsysWarningHandler();
//------------------------------------------------------------------------------------------------------
//------------------------------ Calculate global error flag  ------------------------------------------  
//------------------------------------------------------------------------------------------------------
xError := bCoresysError OR bSubsysError;
xWarning := bSubsysWarning;
END_METHOD

METHOD M_SubsysErrorHandle
VAR_INPUT
END_VAR
VAR
	udiLoop : UDINT;
END_VAR
VAR_OUTPUT
	xError : BOOL;
END_VAR
IF bMachineCtrlInitDOne THEN
	FOR udiLoop := 1 TO cudiXTS_MaxIndex DO
		IF arAlarmHandleValid[udiLoop] = E_AlarmHandleValid.Valid THEN
			arFB_SubsysErrorScan[udiLoop](xSubPMLa := PackTags.arrSubSys_Station^[udiLoop].Admin,
										xUnitName := CONCAT('ST', UDINT_TO_STRING(udiLoop)),
										xUnitID := UDINT_TO_DINT(udiLoop));
		END_IF
	END_FOR
END_IF

bST01_Alarm := (arFB_SubsysErrorScan[1].uiCurrentAlarmsCount > 0);
bST03_Alarm := (arFB_SubsysErrorScan[3].uiCurrentAlarmsCount > 0);
bST06_Alarm := (arFB_SubsysErrorScan[6].uiCurrentAlarmsCount > 0);
bST10_Alarm := (arFB_SubsysErrorScan[10].uiCurrentAlarmsCount > 0);
bST12_Alarm := (arFB_SubsysErrorScan[12].uiCurrentAlarmsCount > 0);
bST14_Alarm := (arFB_SubsysErrorScan[14].uiCurrentAlarmsCount > 0);
bST15_Alarm := (arFB_SubsysErrorScan[15].uiCurrentAlarmsCount > 0);
bST17_Alarm := (arFB_SubsysErrorScan[17].uiCurrentAlarmsCount > 0);
bST18_Alarm := (arFB_SubsysErrorScan[18].uiCurrentAlarmsCount > 0);
bST20_Alarm := (arFB_SubsysErrorScan[20].uiCurrentAlarmsCount > 0);
bST22_Alarm := (arFB_SubsysErrorScan[22].uiCurrentAlarmsCount > 0);
bST23_Alarm := (arFB_SubsysErrorScan[23].uiCurrentAlarmsCount > 0);
bST25_Alarm := (arFB_SubsysErrorScan[25].uiCurrentAlarmsCount > 0);
bST27_Alarm := (arFB_SubsysErrorScan[27].uiCurrentAlarmsCount > 0);
bST30_Alarm := (arFB_SubsysErrorScan[30].uiCurrentAlarmsCount > 0);

xError := bST01_Alarm
	OR bST03_Alarm
	OR bST06_Alarm
	OR bST10_Alarm
	OR bST12_Alarm
	OR bST14_Alarm
	OR bST15_Alarm
	OR bST17_Alarm
	OR bST18_Alarm
	OR bST20_Alarm
	OR bST22_Alarm
	OR bST23_Alarm
	OR bST25_Alarm
	OR bST27_Alarm
	OR bST30_Alarm;
END_METHOD

METHOD M_SubsysWarningHandler
VAR_INPUT
END_VAR

VAR
	udiLoop: UDINT;
END_VAR
IF bMachineCtrlInitDOne THEN
	FOR udiLoop := 1 TO cudiXTS_MaxIndex DO
		arrUnitsWarningHandler[udiLoop]();
		IF arAlarmHandleValid[udiLoop] = E_AlarmHandleValid.Valid THEN
			I_UnitsWarningHandler[udiLoop] := arrUnitsWarningHandler[udiLoop];
			I_UnitsWarningHandler[udiLoop].SetUnitWarningList := (PackTags.arrSubSys_Station^[udiLoop].Admin.Warning );
			I_UnitsWarningHandler[udiLoop].SetUnitID := UDINT_TO_DINT(udiLoop);
			I_UnitsWarningHandler[udiLoop].SetUnitName := CONCAT('ST', UDINT_TO_STRING(udiLoop));
		END_IF
	END_FOR
	bSubsysWarning := FALSE;
	FOR udiLoop := 1 TO cudiXTS_MaxIndex DO
		IF arAlarmHandleValid[udiLoop] = E_AlarmHandleValid.Valid THEN
			IF  I_UnitsWarningHandler[udiLoop].GetWarningStatus THEN
				bSubsysWarning := TRUE;
			END_IF
		END_IF
	END_FOR
END_IF
END_METHOD

METHOD M_SubsysWarrningHandle
VAR_INPUT
END_VAR

VAR
	udiLoop : UDINT;
END_VAR
VAR_INST
	bST30_EmphtyCheck_NG1 : BOOL;
	bST30_EmphtyCheck_NG2 : BOOL;
	bST30_EmphtyCheck_NG3 : BOOL;
	bST30_EmphtyCheck_NG4 : BOOL;
END_VAR
VAR_OUTPUT
	xWarning : BOOL;
END_VAR
IF bMachineCtrlInitDOne THEN
//	FOR udiLoop := 1 TO cudiXTS_MaxIndex DO
//		IF arAlarmHandleValid[udiLoop] = E_AlarmHandleValid.Valid THEN
//			arFB_WarrningHandler[udiLoop](xSubPMLa := PackTags.arrSubSys_Station^[udiLoop].Admin,
//											xUnitName := CONCAT('ST', UDINT_TO_STRING(udiLoop)),
//											xUnitID := UDINT_TO_DINT(udiLoop));
//		END_IF
//	END_FOR
END_IF

bST30_EmphtyCheck_NG1 := FUN_ObserverWarning(xErrorID := 200, xUnitID := 30);
bST30_EmphtyCheck_NG2 := FUN_ObserverWarning(xErrorID := 201, xUnitID := 30);
bST30_EmphtyCheck_NG3 := FUN_ObserverWarning(xErrorID := 202, xUnitID := 30);
bST30_EmphtyCheck_NG4 := FUN_ObserverWarning(xErrorID := 203, xUnitID := 30);
END_METHOD

METHOD M_UploadData
VAR_INPUT
END_VAR
M_UploadTriggerData();
M_UploadResetData();
END_METHOD

METHOD PRIVATE M_UploadResetData : BOOL
VAR_INPUT
END_VAR
VAR_INST
	iStep : INT;
	stAlarm	: ST_Alarm_WString;
	stAlarmInf_DB: ST_AlarmInfo_DB;
END_VAR
CASE iStep OF
	0:
		IF 			fbAlarmResetList.udiGetQueuedAmount <> 0 // Queue裡面有資料
		AND_THEN 	fbAlarmResetList.readElementbyIndex(udiIndex := 1,	pbtReadElement := ADR(stAlarm),	udiReadSize := SIZEOF(stAlarm),	uiErrorID =>) THEN
			
			iStep := iStep + 100;
		END_IF
	
	100:
		stAlarmInf_DB.diMsgNumber := stAlarm.ID;
		stAlarmInf_DB.iMsgClass := stAlarm.eMsgClass;
		stAlarmInf_DB.iMsgProc := 1;
		stAlarmInf_DB.iStateAfter := 0;
		stAlarmInf_DB.sPLC := 'CoreSystem';
		stAlarmInf_DB.sTimeString := FUN_DateTime_To_TMaxString(DateTime := stAlarm.ackDateTime);
		stAlarmInf_DB.wsMsgText := stAlarm.Message;
		
		IF NOT Global_DataFlow.bDataFlowTestByLeo THEN
			IF FB_DataUpload.M_AddAlarmHistory(stAlarmInfo := stAlarmInf_DB) THEN
				iStep := iStep + 100;
			END_IF
		ELSE
			(* Add alarm history to database *)
//			IF Global_DataFlow.fbDataBaseManagement.M_Add_AlarmHistory(addData := stAlarmInf_DB) THEN
//				iStep := iStep + 100;
//			END_IF
		END_IF
	
	200:
		IF fbAlarmResetList.dequeueElement(pbtDequeueElement := ADR(stAlarm),
														udiDequeueSize := SIZEOF(stAlarm),
														uiErrorID =>)
			THEN // 清除已經上傳的資料
			iStep := 0;
		END_IF
		
END_CASE
END_METHOD

METHOD PRIVATE M_UploadTriggerData : BOOL
VAR_INPUT
END_VAR
VAR_INST
	iStep : INT;
	stAlarm	: ST_Alarm_WString;
	stAlarmInf_DB: ST_AlarmInfo_DB;
END_VAR
CASE iStep OF
	0:
		IF 			fbAlarmTrigList.udiGetQueuedAmount <> 0 // Queue裡面有資料
		AND_THEN 	fbAlarmTrigList.readElementbyIndex(udiIndex := 1,	pbtReadElement := ADR(stAlarm),	udiReadSize := SIZEOF(stAlarm),	uiErrorID =>) THEN
			
			iStep := iStep + 100;
		END_IF
	
	100:
		stAlarmInf_DB.diMsgNumber := stAlarm.ID;
		stAlarmInf_DB.iMsgClass := stAlarm.eMsgClass;
		stAlarmInf_DB.iMsgProc := 1;
		stAlarmInf_DB.iStateAfter := 1;
		stAlarmInf_DB.sPLC := 'CoreSystem';
		stAlarmInf_DB.sTimeString := FUN_DateTime_To_TMaxString(DateTime := stAlarm.DateTime);
		stAlarmInf_DB.wsMsgText := stAlarm.Message;
		
		IF NOT Global_DataFlow.bDataFlowTestByLeo THEN
			IF FB_DataUpload.M_AddAlarmHistory(stAlarmInfo := stAlarmInf_DB) THEN
				iStep := iStep + 100;
			END_IF
		ELSE
			IF Global_DataFlow.fbDataBaseManagement.M_Add_AlarmHistory(addData := stAlarmInf_DB) THEN
				iStep := iStep + 100;
			END_IF
		END_IF
		
	200:
		IF fbAlarmTrigList.dequeueElement(pbtDequeueElement := ADR(stAlarm),
														udiDequeueSize := SIZEOF(stAlarm),
														uiErrorID =>)
			THEN // 清除已經上傳的資料
			iStep := 0;
		END_IF
		
END_CASE
END_METHOD

METHOD M_XTSErrorHandle
VAR_INPUT
END_VAR
FB_XTSErrorHandler(xSubPMLa := PackTags.XTS.Admin, xUnitName := 'XTS', xUnitID := 99,xError=>bXTSError);
END_METHOD

END_FUNCTION_BLOCK

// ---- Library/99_Utilities/FB_XY_Move.TcPOU
(* This FB is use to controll two axis to gear in move at the same time 
*)
FUNCTION_BLOCK FB_XY_Move EXTENDS FB_ActionBasic
VAR_INPUT
	xExecute : BOOL;
	xAbort : BOOL;
	xReset :BOOL;
	AxisX_No : AxisNo;
	AxisY_No : AxisNo;
	
    TimeOut     : LREAL := 30; // Unit : s
END_VAR
VAR_OUTPUT
	xAborted : BOOL;
END_VAR
VAR
	StateBehavior : CBML.ETrigATo;
	CurrentPosData :ST_PositionTable;
	uiCyclicStep :UINT;
END_VAR

THIS^.IBehaviourModel := StateBehavior;
StateBehavior(xExecute := xExecute,
              xAbort := xAbort,
              udiTimeOut := LREAL_TO_UDINT(TimeOut * 1000000),
              xDone => xDone,
              xBusy => xBusy,
              xError => xError,
              xAborted => xAborted);

METHOD CleanupAction
VAR_INPUT
    xAbortProposed : BOOL;
    iErrorIDProposed: INT;
END_VAR
VAR_OUTPUT
    xComplete : BOOL := TRUE;
    xAbort: BOOL := xAbortProposed;
 	iErrorID : INT := iErrorIDProposed;
END_VAR
END_METHOD

METHOD CyclicAction
VAR_INPUT
    itfTimingController : CBML.ITimingController;
END_VAR
VAR_OUTPUT
    xComplete : BOOL := TRUE;
    iErrorID : INT := 0;
END_VAR
xComplete := FALSE;
END_METHOD

METHOD ExitAction
VAR_INPUT
    xAfterCleanup : BOOL;
    xInCopyCode : BOOL;
END_VAR
END_METHOD

METHOD ResetAction
VAR_OUTPUT
    xComplete : BOOL := TRUE;
END_VAR
END_METHOD

METHOD StartAction
VAR_OUTPUT
    xComplete : BOOL := TRUE;
	iErrorID : INT := 0;
END_VAR

VAR_INST
	AxisX_Ready :BOOL;
	AxisY_Ready :BOOL;
END_VAR
xComplete := FALSE;
uiCyclicStep := 0;
AxisX_Ready := FUN_CheckAxisAllowMove(AxisNo := AxisX_No);
AxisY_Ready := FUN_CheckAxisAllowMove(AxisNo := AxisY_No);

IF NOT AxisX_Ready THEN
	iErrorID := 2; // AxisX not ready
ELSIF NOT AxisY_Ready THEN
	iErrorID := 3; // AxisY not Ready
ELSIF AxisX_Ready AND AxisY_Ready THEN
	iErrorID := 0;
	xComplete := TRUE;
END_IF
END_METHOD

END_FUNCTION_BLOCK

// ---- Library/99_Utilities/FUNCTION/FUN_CheckAxisAllowMove.TcPOU
FUNCTION FUN_CheckAxisAllowMove : bool
VAR_INPUT
	AxisNo :AxisNo;
END_VAR
VAR
END_VAR

IF arAxisCtrl_gb[THIS^.AxisNo].Admin.Axis.Status.NotMoving AND NOT arAxisCtrl_gb[THIS^.AxisNo].Admin.Axis.Status.Error THEN
	FUN_CheckAxisAllowMove := TRUE;
ELSE
	FUN_CheckAxisAllowMove := FALSE;
END_IF

END_FUNCTION

// ---- Library/99_Utilities/FB_XY_PickAndPlace.TcPOU
FUNCTION_BLOCK FB_XY_PickAndPlace EXTENDS FB_ActionBasic
VAR_INPUT
	xExecute : BOOL;
	xAbort : BOOL;
	xReset :BOOL;
	AxisX_No : AxisNo;
	AxisY_No : AxisNo;
    TimeOut     : LREAL := 30; // Unit : s

END_VAR
VAR_OUTPUT
	xAborted : BOOL;
END_VAR
VAR
	StateBehavior :CBML.ETrigATo;
	Cylinder : REFERENCE TO UNI_CylinderList;
END_VAR

THIS^.IBehaviourModel := StateBehavior;
StateBehavior(
	xExecute:= xExecute, 
	xAbort:= xAbort, 
	udiTimeOut:= LREAL_TO_UDINT( TimeOut*1000000), 
	xDone=> xDone, 
	xBusy=> xBusy, 
	xError=> xError, 
	xAborted=> xAborted);

METHOD CleanupAction
VAR_INPUT
    xAbortProposed : BOOL;
    iErrorIDProposed: INT;
END_VAR
VAR_OUTPUT
    xComplete : BOOL := TRUE;
    xAbort: BOOL := xAbortProposed;
 	iErrorID : INT := iErrorIDProposed;
END_VAR
END_METHOD

METHOD CyclicAction
VAR_INPUT
    itfTimingController : CBML.ITimingController;
END_VAR
VAR_OUTPUT
    xComplete : BOOL := TRUE;
    iErrorID : INT := 0;
END_VAR
END_METHOD

METHOD ExitAction
VAR_INPUT
    xAfterCleanup : BOOL;
    xInCopyCode : BOOL;
END_VAR
END_METHOD

METHOD ResetAction
VAR_OUTPUT
    xComplete : BOOL := TRUE;
END_VAR
END_METHOD

METHOD StartAction
VAR_OUTPUT
    xComplete : BOOL := TRUE;
	iErrorID : INT := 0;
END_VAR
IF
END_METHOD

END_FUNCTION_BLOCK

// ---- Library/99_Utilities/FUNCTION/FUN_ResetStorageCylinder.TcPOU
FUNCTION FUN_ResetStorageCylinder : BOOL
VAR_INPUT
END_VAR
VAR
END_VAR

END_FUNCTION

// ---- Library/99_Utilities/FUNCTION/FUN_RetractStorageCylinder.TcPOU
FUNCTION FUN_RetractStorageCylinder : BOOL
VAR_INPUT
END_VAR
VAR
END_VAR

END_FUNCTION

// ---- POUs/CheckProg/CheckBounds.TcPOU
// Implicitly generated code : DO NOT EDIT
FUNCTION CheckBounds : DINT
VAR_INPUT
	index, lower, upper: DINT;
END_VAR

// Implicitly generated code : Only an Implementation suggestion
{noflow}
IF  index < lower THEN
	CheckBounds := lower;
ELSIF  index > upper THEN
	CheckBounds := upper;
ELSE  
	CheckBounds := index;
END_IF
{flow}

END_FUNCTION

// ---- POUs/CheckProg/CheckDivDInt.TcPOU
// Implicitly generated code : DO NOT EDIT
FUNCTION CheckDivDInt : DINT
VAR_INPUT
	divisor:DINT;
END_VAR

// Implicitly generated code : Only an Implementation suggestion
{noflow}
IF divisor = 0 THEN
	CheckDivDInt:=1;
ELSE
	CheckDivDInt:=divisor;
END_IF;
{flow}

END_FUNCTION

// ---- POUs/CheckProg/CheckDivLInt.TcPOU
// Implicitly generated code : DO NOT EDIT
FUNCTION CheckDivLInt : LINT
VAR_INPUT
	divisor:LINT;
END_VAR

// Implicitly generated code : Only an Implementation suggestion
{noflow}
IF divisor = 0 THEN
	CheckDivLInt:=1;
ELSE
	CheckDivLInt:=divisor;
END_IF;
{flow}

END_FUNCTION

// ---- POUs/CheckProg/CheckDivLReal.TcPOU
// Implicitly generated code : DO NOT EDIT
FUNCTION CheckDivLReal : LREAL
VAR_INPUT
	divisor:LREAL;
END_VAR

// Implicitly generated code : Only an Implementation suggestion
{noflow}
IF divisor = 0 THEN
	CheckDivLReal:=1;
ELSE
	CheckDivLReal:=divisor;
END_IF;
{flow}

END_FUNCTION

// ---- POUs/CheckProg/CheckDivReal.TcPOU
// Implicitly generated code : DO NOT EDIT
FUNCTION CheckDivReal : REAL
VAR_INPUT
	divisor:REAL;
END_VAR

// Implicitly generated code : Only an Implementation suggestion
{noflow}
IF divisor = 0 THEN
	CheckDivReal:=1;
ELSE
	CheckDivReal:=divisor;
END_IF;
{flow}

END_FUNCTION

// ---- POUs/CheckProg/CheckLRangeSigned.TcPOU
// Implicitly generated code : DO NOT EDIT
FUNCTION CheckLRangeSigned : LINT
VAR_INPUT
	value, lower, upper: LINT;
END_VAR

// Implicitly generated code : Only an Implementation suggestion
{noflow}
IF (value < lower) THEN
	CheckLRangeSigned := lower;
ELSIF(value > upper) THEN
	CheckLRangeSigned := upper;
ELSE
	CheckLRangeSigned := value;
END_IF

{flow}

END_FUNCTION

// ---- POUs/CheckProg/CheckLRangeUnsigned.TcPOU
// Implicitly generated code : DO NOT EDIT
FUNCTION CheckLRangeUnsigned : ULINT
VAR_INPUT
	value, lower, upper: ULINT;
END_VAR

// Implicitly generated code : Only an Implementation suggestion
{noflow}
IF (value < lower) THEN
	CheckLRangeUnsigned := lower;
ELSIF(value > upper) THEN
	CheckLRangeUnsigned := upper;
ELSE
	CheckLRangeUnsigned := value;
END_IF
{flow}

END_FUNCTION

// ---- POUs/CheckProg/CheckPointer.TcPOU
// Implicitly generated code : DO NOT EDIT
FUNCTION CheckPointer : POINTER TO BYTE
VAR_INPUT 
	ptToTest : POINTER TO BYTE; // Destination address of the pointer
	iSize : DINT;		        // Size of the type the pointer points to. (e.g: 20 for POINTER TO ARRAY [0..9] OF INT) 
	iGran : DINT;		        // Granularity of the pointer access. This is the size of the biggest non-structured data type in the type the pointer points to. (e.g: 2 for POINTER TO ARRAY [0..9] OF INT)
	bWrite: BOOL;		        // Indicates read or write Access. TRUE = write access.
END_VAR

// Implicitly generated code : Only an Implementation suggestion
{noflow}
IF ptToTest=0 THEN
    ADSLOGSTR(ADSLOG_MSGTYPE_ERROR OR ADSLOG_MSGTYPE_STRING,'CheckPointer failed due to invalid address.','');
ELSIF iSize<=0 THEN
    ADSLOGSTR(ADSLOG_MSGTYPE_ERROR OR ADSLOG_MSGTYPE_STRING,'CheckPointer failed due to invalid size.','');
ELSIF iGran<=0 THEN
    ADSLOGSTR(ADSLOG_MSGTYPE_ERROR OR ADSLOG_MSGTYPE_STRING,'CheckPointer failed due to invalid granularity.','');
// -> Please note that the following memory area check is time consuming:
//ELSIF F_CheckMemoryArea(pData:=ptToTest,nSize:=DINT_TO_UDINT(iSize)) = E_TcMemoryArea.Unknown THEN
//    ADSLOGSTR(ADSLOG_MSGTYPE_ERROR OR ADSLOG_MSGTYPE_STRING,'CheckPointer failed due to unknown memory area.','');
END_IF
CheckPointer := ptToTest;
{flow}

END_FUNCTION

// ---- POUs/CheckProg/CheckRangeSigned.TcPOU
// Implicitly generated code : DO NOT EDIT
FUNCTION CheckRangeSigned : DINT
VAR_INPUT
	value, lower, upper: DINT;
END_VAR

// Implicitly generated code : Only an Implementation suggestion
{noflow}
IF (value < lower) THEN
	CheckRangeSigned := lower;
ELSIF(value > upper) THEN
	CheckRangeSigned := upper;
ELSE
	CheckRangeSigned := value;
END_IF
{flow}

END_FUNCTION

// ---- POUs/CheckProg/CheckRangeUnsigned.TcPOU
// Implicitly generated code : DO NOT EDIT
FUNCTION CheckRangeUnsigned : UDINT
VAR_INPUT
	value, lower, upper: UDINT;
END_VAR

// Implicitly generated code : Only an Implementation suggestion
{noflow}
IF (value < lower) THEN
	CheckRangeUnsigned := lower;
ELSIF(value > upper) THEN
	CheckRangeUnsigned := upper;
ELSE
	CheckRangeUnsigned := value;
END_IF
{flow}

END_FUNCTION
